// TwinCAT 3 PLC project FlyingSaw
// ProgramVersion: 3.1.4024.0
// libraries:
//   Tc2_MC2, * (Beckhoff Automation GmbH)
//   Tc2_MC2_FlyingSaw, * (Beckhoff Automation GmbH)
//   Tc2_NC, * (Beckhoff Automation GmbH)
//   Tc2_Standard, * (Beckhoff Automation GmbH)
//   Tc2_System, * (Beckhoff Automation GmbH)
//   Tc3_Module, * (Beckhoff Automation GmbH)
// project tree:
//   / GlobalTextList.TcGTLO, PlcTask.TcTTO, Visualization Manager.TcVMO (not stored)
//   POUs/ AxisSync.TcPOU, FlyingSaw.TcPOU, MAIN.TcPOU, State.TcDUT, Visualization.TcVIS

CONFIGURATION FlyingSaw
    RESOURCE PLC ON TwinCAT3
        TASK PlcTask(INTERVAL := T#10ms, PRIORITY := 20);
        PROGRAM MAIN WITH PlcTask : MAIN;
    END_RESOURCE
END_CONFIGURATION

// ---- POUs/State.TcDUT
{attribute 'qualified_only'}
{attribute 'strict'}
TYPE State :
(
	CheckEnable := 0,
	Initialize := 5,
	WaitForButton := 10,
	StartMaster := 20,
	Synchronization := 30,
	FinishAndStopMotors := 40,
	GearOut := 50,
	ErrorState := 999
	
);
END_TYPE

// ---- POUs/MAIN.TcPOU
PROGRAM MAIN
VAR
END_VAR

FlyingSaw(); //we call the program

END_PROGRAM

// ---- POUs/FlyingSaw.TcPOU
PROGRAM FlyingSaw
VAR
	fbAxisSync : AxisSync; //we initialize the function block that does all the logic
	
	bReset : BOOL; //bool variable connected to a button in the HMI
	bMove : BOOL; //bool variable connected to a button in the HMI
	
	bSensor : BOOL; //bool variable connected to a light in the HMI (turns on when the sync process starts)
	
	rMasterPosition : LREAL; //LREAL variables that display the position of the motors
	rSlavePosition : LREAL;
END_VAR

fbAxisSync.bButton := bMove; //we connect all the variables to the variables of the function block accordingly
fbAxisSync.bResetButton := bReset;

bSensor := fbAxisSync.bSyncSensor;

rMasterPosition := fbAxisSync.rMasterPos;
rSlavePosition := fbAxisSync.rSlavePos;

fbAxisSync(); //we call the funciton block

END_PROGRAM

// ---- POUs/AxisSync.TcPOU
FUNCTION_BLOCK AxisSync
VAR_INPUT
	bButton : BOOL; //button which the user can press to start the master motor
	bResetButton : BOOL; //button to reset the axis incase an error occurs
END_VAR
VAR_OUTPUT
	bSyncSensor : BOOL; //sensor that turns on a light when the sync process starts
	rMasterPos : LREAL; //sensor that displays the position of the master
	rSlavePos : LREAL; //sensor that displays the position of the slave
END_VAR
VAR
	iState : State; 
	
	MasterMotor : AXIS_REF; //master motor instance
	SlaveMotor : AXIS_REF; //slave motor instance
	
	PowerMaster : MC_Power; //motion function blocks for the master
	ResetMaster : MC_Reset;
	MoveMaster : MC_MoveAbsolute;
	JogMaster : MC_Jog;
	StopMaster : MC_Stop;
	
	PowerSlave : MC_Power; //motion function blocks for the slave
	ResetSlave : MC_Reset;
	MoveSlave : MC_MoveAbsolute;
	JogSlave : MC_Jog;
	StopSlave : MC_Stop;
	
	FlyingSaw : MC_GearInPos; //sync function block
	GearOut : MC_GearOut; //gear out function block
	
	TimerSync : TON; //timer that gets enabled and starts the sync process
END_VAR

CASE iState OF
	State.CheckEnable: //we check whether the motors are ON	
		IF PowerMaster.Enable AND PowerSlave.Enable THEN
			iState := State.Initialize;
		END_IF
	State.Initialize: //initialization state (we reset the timers,reset the motion function blocks and we set the motors to position 0)	
		TimerSync.IN := FALSE;
		
		StopMaster(Axis := MasterMotor,Execute := FALSE);
		StopSlave(Axis := SlaveMotor,Execute := FALSE);
		
		ResetMaster(Axis := MasterMotor,Execute := FALSE);
		ResetSlave(Axis := SlaveMotor,Execute := FALSE);
		
		MoveMaster(Axis := MasterMotor,Position := 0,Velocity := 100,Execute := TRUE); //move the motors to position 0
		MoveSlave(Axis := SlaveMotor,Position := 0,Velocity := 100,Execute := TRUE);
		
		IF NOT MoveMaster.Busy AND NOT MoveSlave.Busy THEN
			MoveMaster(Axis := MasterMotor,Execute := FALSE); //when we finish moving them reset the function blocks as well
			MoveSlave(Axis := SlaveMotor,Execute := FALSE);
			iState := State.WaitForButton;
		END_IF		
	State.WaitForButton: //in this state we wait for the user to start the master motor
		IF bButton THEN
			iState := State.StartMaster;
		END_IF
	State.StartMaster: //here we move the master motor to position 1440
		IF NOT MoveMaster.Error THEN
			MoveMaster(Axis := MasterMotor,Position := 1440,Velocity := 70,Execute := TRUE);
			iState := State.Synchronization;
		ELSE
			iState := State.ErrorState; //if an error occurs go to the error state
		END_IF
	State.Synchronization: //start the sync process
		TimerSync.IN := TRUE;  //enable the timer
		IF TimerSync.Q THEN //after the ET passes activate the sync
			bSyncSensor := TRUE; 
			FlyingSaw(Master := MasterMotor,Slave := SlaveMotor,MasterSyncPosition := 540,SlaveSyncPosition := 540,Velocity := 500,Execute := TRUE);
			iState := State.FinishAndStopMotors;
		END_IF
		IF MoveMaster.Error THEN //if an error occurs go to the error state
			iState := State.ErrorState;
		END_IF
	State.FinishAndStopMotors: //when the master motor reaches the desired position stop the motors and go to the ger out state
		FlyingSaw(Master := MasterMotor,Slave := SlaveMotor,Execute := FALSE); //reset this function block
		IF MoveMaster.Done THEN
			StopMaster(Axis := MasterMotor,Deceleration := 300,Execute := TRUE);
			MoveMaster(Axis := MasterMotor,Execute := FALSE);
			bSyncSensor := FALSE;
			iState := State.GearOut;
		ELSIF MoveMaster.Error THEN //if an error occurs go to the error handling state
			iState := State.ErrorState;
		END_IF
	State.GearOut:
		GearOut(Slave := SlaveMotor,Execute := TRUE); //we gear out the motors and reset the function block
		IF GearOut.Done THEN
			GearOut(Slave := SlaveMotor,Execute := FALSE);
			iState := State.CheckEnable; //return to the start
		END_IF
	State.ErrorState: //error handling state
		bSyncSensor := FALSE;
		StopMaster(Axis := MasterMotor,Deceleration := 300,Execute := TRUE); //if an error occurs we stop the motors
		StopSlave(Axis := SlaveMotor,Deceleration := 300,Execute := TRUE);
		IF bResetButton	THEN //wait for the error to be resolved and if the reset button is pressed reset the motors and return to the start
			ResetMaster(Axis := MasterMotor,Execute := TRUE);
			ResetSlave(Axis := SlaveMotor,Execute := TRUE);
			MoveMaster(Axis := MasterMotor,Execute := FALSE);
			MoveSlave(Axis := SlaveMotor,Execute := FALSE);
			iState := State.CheckEnable;
		END_IF
		
END_CASE

PowerMaster(Axis := MasterMotor,Enable := TRUE,Enable_Positive := TRUE,Enable_Negative := TRUE);
ResetMaster(Axis := MasterMotor);
MoveMaster(Axis := MasterMotor);
JogMaster(Axis := MasterMotor);
StopMaster(Axis := MasterMotor);

PowerSlave(Axis := SlaveMotor,Enable := TRUE,Enable_Positive := TRUE,Enable_Negative := TRUE);
ResetSlave(Axis := SlaveMotor);
MoveSlave(Axis := SlaveMotor);
JogSlave(Axis := SlaveMotor);
StopSlave(Axis := SlaveMotor);

rMasterPos := MasterMotor.NcToPlc.ActPos;
rSlavePos := SlaveMotor.NcToPlc.ActPos;

TimerSync(PT := T#6000MS);

END_FUNCTION_BLOCK

// ---- GlobalTextList.TcGTLO
TEXTLIST GlobalTextList
  928 = 'Reset Axis'
  230 = 'Start Master'
  840 = 'Start Sync'
END_TEXTLIST

// ---- POUs/Visualization.TcVIS
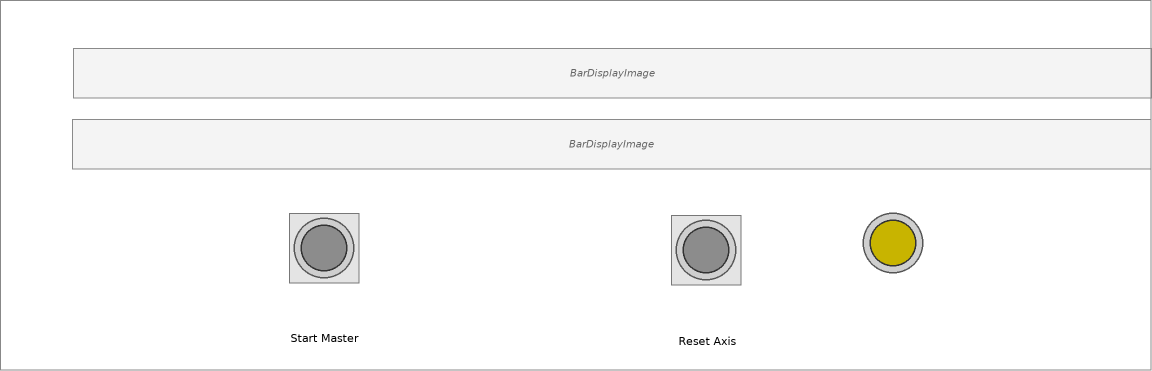
VISUALIZATION Visualization  // 1152x371
    PushSwitch (289,213 70x70), variable: FlyingSaw.bMove, behaviour: TAP, style: Switch-PushSwitch-Gray
    PushSwitch (671,215 70x70), variable: FlyingSaw.bReset, behaviour: TAP, style: Switch-PushSwitch-Gray
    Lamp1 (858,208 70x70), variable: FlyingSaw.bSensor, style: Lamp-Lamp1-Yellow
    BarDisplayImage (73,48 1079x50), value: FlyingSaw.rMasterPosition, style: BarDisplayImage-Gray, scale format: %.1f, scale 0..1440
    BarDisplayImage (72,119 1079x50), value: FlyingSaw.rSlavePosition, style: BarDisplayImage-Gray, scale format: %.1f, scale 0..1440
    Label (240,309 169x59), "Start Master"
    Label (623,312 169x59), "Reset Axis"
END_VISUALIZATION
